FUNCTION_BLOCK FB_SIM_Fuellstand
VAR_INPUT
	I_Fuellen			:BOOL;
END_VAR

VAR_OUTPUT
	O_SensorSignal		:INT;
END_VAR
	
VAR
	V_Delay				:TON;
	V_TimeStatus		:BOOL;
END_VAR

// Timer instanziieren
V_Delay(IN := V_TimeStatus, PT := T#1S);	

IF I_Fuellen THEN
	// Grundwert definieren
	O_SensorSignal := 0;
	
	// Timer starten
	V_TimeStatus := TRUE;
	
	// Reaktor füllen
	IF V_Delay.Q THEN
		V_TimeStatus := FALSE;
		O_SensorSignal := O_SensorSignal + (27648/100);
	END_IF
END_IF

END_FUNCTION_BLOCK

(* stored: Version 1.1.0.1, ProductVersion 3.1.4024.12
   POU FB_SIM_Fuellstand: Id {73040a9e-8d81-4131-9405-ae552231ddca}, SpecialFunc None *)
